{attribute 'GeneratedUsingTerminal: KL1352'}
{attribute addProperty BoxType "KL1352"}
{attribute addProperty Id "InputAT %I*BOOL0ErrorAT %I*BOOL0"}
{attribute addProperty CRC "584898197"}
{attribute addProperty Size "0"}
TYPE Channel_22DCD695 :
STRUCT
	{attribute addProperty Name "Input"}
	Input AT %I* : BOOL;
	{attribute addProperty Name "Error"}
	Error AT %I* : BOOL;
END_STRUCT
END_TYPE
